FUNCTION_BLOCK AnalogInput EXTENDS BaseIO
VAR_INPUT
	ProcessValue: LREAL;
	Override: BOOL;
	OverrideValue: LREAL;
END_VAR
VAR_OUTPUT
	Value: LREAL;
END_VAR
VAR
	InitDone: BOOL;
	TempValue: LREAL;
END_VAR
VAR PERSISTENT
	SignedWord: BOOL;
	ProcessMin: DINT := 0;
	ProcessMax: DINT := 16#3FFF;
	MinValue: LREAL := 0;
	MaxValue: LREAL := 1;
	SavedOverride: BOOL;
	SavedOverrideValue: LREAL;
END_VAR

SUPER^();
IF NOT InitDone THEN
	InitDone := TRUE;
	OverrideValue := SavedOverrideValue;
	Override := SavedOverride;	
END_IF
IF NOT Override THEN
	TempValue := ProcessValue;
	IF SignedWord THEN
		IF ProcessValue >= 16#8000 THEN
			TempValue := TempValue - 16#10000;
		END_IF
	END_IF
	Value := GetValue();
	Error := ProcessError;
	ErrorCode := ProcessErrorCode;
ELSE
	Value := OverrideValue;
	Error := FALSE;
	ErrorCode := 0;
END_IF
SavedOverride := Override;
SavedOverrideValue := OverrideValue;

METHOD GetValue : LREAL
VAR_INPUT
END_VAR
GetValue := (LimitValue(TempValue, ProcessMin, ProcessMax) - ProcessMin) / (ProcessMax - ProcessMin) * (MaxValue - MinValue) + MinValue;
END_METHOD

END_FUNCTION_BLOCK

(* stored: Version 1.1.0.1, ProductVersion 3.1.4024.6
   POU AnalogInput: Id {1d1cb0c1-c0d3-4db6-a9bb-1f03a14e198d}, SpecialFunc None
   Method GetValue: Id {910725f1-c0fb-409c-a151-64f03276bf5f} *)
